// TIA Portal V17 export
FUNCTION "FC_烧嘴报警" : Void   // FC, LAD
{ S7_Optimized_Access := 'TRUE' }
BEGIN
END_FUNCTION
